TYPE
    ColorsSignalLightMachineModes :
    STRUCT
        Green       : BOOL;
        Yellow      : BOOL;
        Red         : BOOL;
    END_STRUCT
END_TYPE

(* stored: Version 1.1.0.1, ProductVersion 3.1.4024.12
   DUT ColorsSignalLightMachineModes: Id {1591cb05-60ac-025a-34bc-1b49e3106441} *)
